// TwinCAT 3 PLC project ModBusPLC
// ProgramVersion: 3.1.4026.9
// libraries:
//   ModBus_For_FactoryIO, * (Kristian Zitny)
//   Tc2_ModbusSrv, * (Beckhoff Automation GmbH)
//   Tc2_Standard, * (Beckhoff Automation GmbH)
//   Tc2_System, * (Beckhoff Automation GmbH)
// project tree:
//   GVLs/ GVL_Factory_IO.TcGVL, GVL_IO.TcGVL
//   / PlcTask.TcTTO
//   POUs/Demonstration/ DemoProgram.TcPOU
//   POUs/Demonstration/DUTS/ E_FIO_PNP_State.TcDUT, ST_FIO_AxisConfig.TcDUT, ST_FIO_AxisIO.TcDUT
//   POUs/Demonstration/FunctionBlocks/ FB_Encoder.TcPOU, FB_FactoryIO_AxisAnalog.TcPOU, FB_FactoryIO_Conveyor.TcPOU, FB_FactoryIO_Lamp.TcPOU, FB_FactoryIO_PickPlace2Axis.TcPOU, FB_FactoryIO_Pusher.TcPOU, FB_Pick_Place.TcPOU, FB_PulseTrain.TcPOU
//   POUs/Factory_IO/ Connection.TcPOU, FB_IOMapper256.TcPOU
//   POUs/ MAIN.TcPOU
// real-time tasks:
//   TASK PlcTask: cycle T#10ms, priority 20, ADS port 350

CONFIGURATION ModBusPLC
    RESOURCE PLC ON TwinCAT3
        TASK PlcTask(INTERVAL := T#10ms, PRIORITY := 20);
        PROGRAM MAIN WITH PlcTask : MAIN;
    END_RESOURCE
END_CONFIGURATION

// ---- POUs/Demonstration/DUTS/E_FIO_PNP_State.TcDUT
TYPE E_FIO_PNP_State :
(
    Idle,
    MoveToPick,
    Grab,
    LiftAfterPick,
    MoveToPlace,
    Release,
    RetractAfterPlace,
    Error
);
END_TYPE

// ---- POUs/Demonstration/DUTS/ST_FIO_AxisConfig.TcDUT
TYPE ST_FIO_AxisConfig :
STRUCT
    MinPos     : LREAL;    // engineering units (e.g. mm)
    MaxPos     : LREAL;    // engineering units
    Tolerance  : LREAL;    // within tolerance -> in position
    Kp         : LREAL;    // proportional gain (engineering units per second)
    MaxVel     : LREAL;    // max velocity (engineering units per second)
END_STRUCT
END_TYPE

// ---- POUs/Demonstration/DUTS/ST_FIO_AxisIO.TcDUT
TYPE ST_FIO_AxisIO :
STRUCT
    SetPos : LREAL;   // output: position command to "analog output"
    ActPos : LREAL;   // input: feedback from "analog input"
END_STRUCT
END_TYPE

// ---- GVLs/GVL_Factory_IO.TcGVL
{attribute 'qualified_only'}
VAR_GLOBAL
	FIOinputs : ARRAY[0..31, 0..7] OF BOOL;
	FIOoutputs : ARRAY [0..255] OF BOOL;
END_VAR

// ---- GVLs/GVL_IO.TcGVL
{attribute 'qualified_only'}
VAR_GLOBAL
	Input : ARRAY [0..255] OF BOOL;
	Output : ARRAY [0..255] OF BOOL;
	AnalogInput : ARRAY [0..63] OF REAL;
	AnalogOutput : ARRAY [0..63] OF REAL;
END_VAR

// ---- POUs/MAIN.TcPOU
PROGRAM MAIN
VAR

END_VAR

// Call Connection Program for Connection with Factory IO Modbus Server //
Connection();
// Call Demo Program
DemoProgram();

END_PROGRAM

// ---- POUs/Factory_IO/Connection.TcPOU
PROGRAM Connection
VAR
	MB_Client: ModBus_For_Factory_IO;
	IO_Mapper: FB_IOMapper256;
END_VAR


	MB_Client(
	axInputs:= GVL_Factory_IO.FIOoutputs, 
	arInputs:= GVL_IO.AnalogOutput, 
	sIPaddr:= '127.0.0.1', 
	uiTCPPort:= 505, 
	iUnitID:= 1, 
	iNumberOfBoolInputs:= 256, 
	iNumberOfRegInputs:= 64, 
	iNumberOfBoolOutputs:= 256, 
	iNumberOfRegOutputs:= 64, 
	xStart:= TRUE, 
	axReaded=> GVL_Factory_IO.FIOinputs, 
	arReaded=> GVL_IO.AnalogInput, 
	xErrReadBoolFB=> , 
	udiErrNumberReadBoolFB=> , 
	sErrorDescriptionReadBoolFB=> , 
	xErrReadRegFB=> , 
	udiErrNumberReadRegFB=> , 
	sErrorDescriptionReadRegFB=> , 
	xErrWriteBoolFB=> , 
	udiErrNumberWriteBoolFB=> , 
	sErrorDescriptionWriteBoolFB=> , 
	xErrWriteRegFB=> , 
	udiErrNumberWriteRegFB=> , 
	sErrorDescriptionWriteRegFB=> );
	
	
	
	IO_Mapper(inputs:= GVL_Factory_IO.FIOinputs, outputs:= GVL_Factory_IO.FIOOutputs );

END_PROGRAM

// ---- POUs/Factory_IO/FB_IOMapper256.TcPOU
FUNCTION_BLOCK FB_IOMapper256
VAR_INPUT
    // Globale IO arrays
    inputs  : ARRAY [0..31, 0..7] OF BOOL;
END_VAR

VAR_IN_OUT
    outputs : ARRAY [0..255] OF BOOL;
END_VAR

VAR_OUTPUT
    
END_VAR

VAR
    i, j     : INT;
    flatIndex: INT;
END_VAR


// ===========================
// 1) Inputs 2D -> flat 0..255
// ===========================
FOR i := 0 TO 31 DO
    FOR j := 0 TO 7 DO
        flatIndex := i * 8 + j;
        GVL_IO.input[flatIndex] := inputs[i, j];
    END_FOR
END_FOR;


// ===========================
// 2) Outputs flat -> global
// ===========================
FOR flatIndex := 0 TO 255 DO
    outputs[flatIndex] := GVL_IO.Output[flatIndex];
END_FOR;

END_FUNCTION_BLOCK

// ---- POUs/Demonstration/DemoProgram.TcPOU
PROGRAM DemoProgram
VAR
	DemoEncoder_1: FB_Encoder;
	DemoEncoder_2: FB_Encoder;
	fEncoder1_Position: LREAL;
	fEncoder1_Velocity: LREAL;
	bEncoder1_Error: BOOL;
	nEncoder1_ErrorID: UINT;
	fEncoder2_Position: LREAL;
	fEncoder2_Velocity: LREAL;
	bEncoder2_Error: BOOL;
	nEncoder2_ErrorID: UINT;
	Start: BOOL;
	 
	ConvLeft: BOOL;
	ConvRight: BOOL;
	RotCW_1: BOOL;
	RotCCW_1: BOOL;
	Grab_1: BOOL;
	ProductSensorBlue: BOOL;
	ProductSensorGreen: BOOL;
	X_Cmd_1: REAL;
	Z_Cmd_1: REAL;
	X_Act_1: REAL;
	Z_Act_1: REAL;
	bXInPos_1: BOOL;
	bZInPos_1: BOOL;
	Sensor_ProductInFrontOfGripper: BOOL;
	LastKnownColour: STRING(INT#4);
	T_Grab_1: TON ;
	T_Rot_1: TON;
	T_Release_1: TON;
	T_EndTimer: TON;
	UseAdvancedMode: BOOL := TRUE;
	T_Rot_0: TON;
	ProductColour: REAL;
	T_Grab_2: TON;
	T_Rot_3: TON;
	T_Rot_4: TON;
	SafeX_1: REAL := 0;
END_VAR
VAR
    // -----------------------------
    // I/O mapping (adjust indices)
    // -----------------------------
    ProductSensor : BOOL;

    ConvAll : BOOL;

    RotCW  : BOOL;
    RotCCW : BOOL;
    Grab   : BOOL;

    // -----------------------------
    // "Analog" feedback/commands
    // -----------------------------
    X_Act : LREAL;
    Z_Act : LREAL;
    X_Cmd : LREAL;
    Z_Cmd : LREAL;

    // -----------------------------
    // Targets (demo values)
    // -----------------------------
    PickX  : LREAL := 6.0;
    PickZ  : LREAL := 10.0;

    PlaceX : LREAL := 7.0;
    PlaceZ : LREAL := 9.0;

    SafeZ  : LREAL := 0.0;
	
	PickX_1  : LREAL := 1.0;
    PickZ_1  : LREAL := 10.0;

    PlaceX_1 : LREAL := 10.0;
    PlaceZ_1 : LREAL := 10.0;

    SafeZ_1  : LREAL := 0.0;

    Tol    : LREAL := 1.0;

    // -----------------------------
    // State machine
    // -----------------------------
    State : INT := 0;
	StateAdvanced : INT := 0;

    // -----------------------------
    // Timers
    // -----------------------------
    T_Grab    : TON;
    T_Release : TON;
    T_Rot     : TON;

    // -----------------------------
    // Rotation pulse control
    // -----------------------------
    RotPulseActive : BOOL;

    // -----------------------------
    // Helpers
    // -----------------------------
    bXInPos : BOOL;
    bZInPos : BOOL;
END_VAR

VAR_INPUT
	
END_VAR

DemoEncoder_1(
	bEnable:= , 
	bA_Input:= GVL_IO.Input[8],
	bB_Input:= GVL_IO.Input[9], 
	bInvertDirection:= , 
	fUnitPerCount:= , 
	nVelSampleMs:= , 
	bRefSensor:= , 
	bRefCommand:= , 
	fRefPosition:= , 
	nCount=> , 
	fPosition=> fEncoder1_Position, 
	fVelocity=> fEncoder1_Velocity, 
	bReferenced=> , 
	bError=> bEncoder1_Error, 
	nErrorId=> nEncoder1_ErrorID);
	
	
	
										// =====================================================
										// Demo Program Simple Pick and Place
										// =====================================================	
		
	// =====================================================
	// Apply outputs (all 3 conveyors together)
	// =====================================================
	GVL_IO.Output[0] := ConvAll;
	GVL_IO.Output[1] := ConvAll;
	GVL_IO.Output[2] := ConvAll;
	GVL_IO.Output[4] := ConvAll;
	// Rotation interlock
	GVL_IO.Output[28] := RotCW ;
	GVL_IO.Output[29] := RotCCW ;
	
	// Grab
	GVL_IO.Output[3] := Grab;
	
	// Analog commands (map these to your Modbus registers / analog outputs)
	GVL_IO.AnalogOutput[0] := LREAL_TO_WORD(X_Cmd ); 
	GVL_IO.AnalogOutput[1] := LREAL_TO_WORD(Z_Cmd );
	

// =====================================================
// Read inputs (adjust mapping here)
// =====================================================
ProductSensor := GVL_IO.Input[7];
X_Act := GVL_IO.AnalogInput[0];
Z_Act := GVL_IO.AnalogInput[1];

// =====================================================
// Default outputs each scan
// =====================================================
//GVL_IO.Output[0] := FALSE; // conveyor 1
//GVL_IO.Output[1] := FALSE; // conveyor 2
//GVL_IO.Output[2] := FALSE; // conveyor 3

//RotCW := FALSE;
//RotCCW := FALSE;
Grab := FALSE;

// Rotation coils default off (interlock)



// Grab output default off
GVL_IO.Output[6] := FALSE; // grab

// Default hold current command
X_Cmd := X_Cmd;
Z_Cmd := Z_Cmd;

IF ConvAll THEN
	GVL_IO.Output[11] := TRUE; //Green Light
	GVL_IO.Output[10]:= FALSE;
	ELSE IF NOT ConvAll THEN
		GVL_IO.Output[10]:= TRUE; //Yellow Light
		GVL_IO.Output[11]:= FALSE;
	END_IF
END_IF

IF Connection.MB_Client.xErrReadBoolFB THEN 
	GVL_IO.Output[9] := TRUE; //Red Light
END_IF
// =====================================================
// Simple in-position checks (needs real feedback)
// =====================================================
bXInPos := (ABS(X_Cmd - X_Act) <= Tol);
bZInPos := (ABS(Z_Cmd - Z_Act) <= Tol);


// =====================================================
// State machine
// =====================================================
CASE State OF

// -----------------------------------------------------
// 0: conveyors on, wait product
// -----------------------------------------------------
0:
    ConvAll := TRUE;

	IF Sensor_ProductInFrontOfGripper THEN
        ConvAll := FALSE;
        State := 110;
    END_IF
	
    IF ProductSensor  THEN
        ConvAll := FALSE;
        State := 10;
    END_IF



// -----------------------------------------------------
// 10: move above pick (SafeZ + PickX)
// -----------------------------------------------------
10:
    ConvAll := FALSE;

    X_Cmd := PickX;
    Z_Cmd := SafeZ;

    IF (ABS(PickX - X_Act) <= Tol) AND (ABS(SafeZ - Z_Act) <= Tol) THEN
        State := 20;
    END_IF


// -----------------------------------------------------
// 20: go down to pick (PickZ)
// -----------------------------------------------------
20:
    ConvAll := FALSE;

    X_Cmd := PickX;
    Z_Cmd := PickZ;

    IF (ABS(PickZ - Z_Act) <= Tol) THEN
        State := 30;
    END_IF


// -----------------------------------------------------
// 30: grab for 0.5s
// -----------------------------------------------------
30:
    ConvAll := FALSE;

    X_Cmd := PickX;
    Z_Cmd := PickZ;

    Grab := TRUE;

    T_Grab(IN := TRUE, PT := T#250ms);
    IF T_Grab.Q THEN
        T_Grab(IN := FALSE);
        State := 40;
    END_IF


// -----------------------------------------------------
// 40: lift to SafeZ (keep grab)
// -----------------------------------------------------
40:
    ConvAll := FALSE;

    X_Cmd := PickX;
    Z_Cmd := SafeZ;

    Grab := TRUE;

    IF (ABS(SafeZ - Z_Act) <= Tol) THEN
        State := 50;
    END_IF


// -----------------------------------------------------
// 50: rotate CW pulse 0.5s (coil 4)
// -----------------------------------------------------
50:
    ConvAll := FALSE;

    X_Cmd := PickX;
    Z_Cmd := SafeZ;

    Grab := TRUE;

    GVL_IO.Output[50] := TRUE;

    T_Rot_0(IN := TRUE, PT := T#1500MS);
    IF T_Rot_0.Q THEN
        T_Rot_0(IN := FALSE);
        State := 60;
    END_IF


// -----------------------------------------------------
// 60: move above place (SafeZ + PlaceX)
// -----------------------------------------------------
60:
    ConvAll := FALSE;
	GVL_IO.Output[50] := FALSE;
    X_Cmd := PlaceX;
    Z_Cmd := SafeZ;

    Grab := TRUE;

    IF (ABS(PlaceX - X_Act) <= Tol) AND (ABS(SafeZ - Z_Act) <= Tol) THEN
        State := 70;
    END_IF


// -----------------------------------------------------
// 70: go down to place (PlaceZ)
// -----------------------------------------------------
70:
    ConvAll := FALSE;

    X_Cmd := PlaceX;
    Z_Cmd := PlaceZ;

    Grab := TRUE;

    IF (ABS(PlaceZ - Z_Act) <= Tol) THEN
        State := 80;
    END_IF


// -----------------------------------------------------
// 80: release and wait 1s
// -----------------------------------------------------
80:
    ConvAll := FALSE;

    X_Cmd := PlaceX;
    Z_Cmd := PlaceZ;

    Grab := FALSE;

    T_Release(IN := TRUE, PT := T#750MS);
    IF T_Release.Q THEN
        T_Release(IN := FALSE);
        State := 90;
    END_IF


// -----------------------------------------------------
// 90: lift again to SafeZ
// -----------------------------------------------------
90:
    ConvAll := FALSE;

    X_Cmd := PlaceX;
    Z_Cmd := SafeZ;

    Grab := FALSE;

    IF (ABS(SafeZ - Z_Act) <= Tol) THEN
        State := 100;
    END_IF


// -----------------------------------------------------
// 100: rotate CCW pulse 0.5s (coil 5)
// -----------------------------------------------------
100:
    ConvAll := FALSE;

    X_Cmd := PlaceX;
    Z_Cmd := SafeZ;

    Grab := FALSE;

    GVL_IO.Output[51] := TRUE;

    T_Rot(IN := TRUE, PT := T#400MS);
    IF T_Rot.Q THEN
        T_Rot(IN := FALSE);
        State := 110;
    END_IF


// -----------------------------------------------------
// 110: conveyors on again, wait sensor clear
// -----------------------------------------------------
110:
	GVL_IO.Output[51] := FALSE;
	IF NOT Sensor_ProductInFrontOfGripper THEN
		ConvAll := TRUE;
	END_IF
    

    IF NOT ProductSensor OR NOT Sensor_ProductInFrontOfGripper THEN
        State := 0;
    END_IF


ELSE
    State := 0;
END_CASE


											// =====================================================
											// Demo Program Advanced Pick and Place
											// =====================================================	
		
	// =====================================================
	// Apply outputs (all 3 conveyors together)
	// =====================================================
	GVL_IO.Output[14] := ConvLeft;
	GVL_IO.Output[15] := ConvLeft;
	GVL_IO.Output[16] := ConvLeft;
	GVL_IO.Output[17] := ConvLeft;
	GVL_IO.Output[18] := ConvLeft;
	GVL_IO.Output[19] := ConvLeft;
	GVL_IO.Output[20] := ConvLeft;
	GVL_IO.Output[21] := ConvRight;
	GVL_IO.Output[22] := ConvRight;
	GVL_IO.Output[23] := ConvRight;
	GVL_IO.Output[24] := ConvRight;
	GVL_IO.Output[25] := ConvRight;
	GVL_IO.Output[26] := ConvRight;
	GVL_IO.Output[27] := ConvRight;
	
	
	// Grab
	GVL_IO.Output[5] := Grab_1;
	
	// Analog commands (map these to your Modbus registers / analog outputs)
	GVL_IO.AnalogOutput[2] := LREAL_TO_WORD(X_Cmd_1 ); 
	GVL_IO.AnalogOutput[3] := LREAL_TO_WORD(Z_Cmd_1 );
	

// =====================================================
// Read inputs (adjust mapping here)
// =====================================================
ProductSensorBlue := GVL_IO.Input[12];
ProductSensorGreen := GVL_IO.Input[13];
Sensor_ProductInFrontOfGripper := GVL_IO.Input[6];
X_Act_1 := GVL_IO.AnalogInput[2];
Z_Act_1 := GVL_IO.AnalogInput[3];
ProductColour := GVL_IO.AnalogInput[4];


// =====================================================
// Default outputs each scan
// =====================================================
//GVL_IO.Output[0] := FALSE; // conveyor 1
//GVL_IO.Output[1] := FALSE; // conveyor 2
//GVL_IO.Output[2] := FALSE; // conveyor 3


Grab_1 := FALSE;
ConvLeft := FALSE;
ConvRight := FALSE;

// Default hold current command
X_Cmd_1 := X_Cmd_1;
Z_Cmd_1 := Z_Cmd_1;


// =====================================================
// Simple in-position checks (needs real feedback)
// =====================================================
bXInPos_1 := (ABS(X_Cmd_1 - X_Act_1) <= Tol);
bZInPos_1 := (ABS(Z_Cmd_1 - Z_Act_1) <= Tol);

// =====================================================
// Colour Helpers
// =====================================================

IF Connection.MB_Client.arReaded[4] = 0.1 THEN
    LastKnownColour := 'BLUE';
ELSIF Connection.MB_Client.arReaded[4] = 5 THEN
    LastKnownColour := 'GREEN';
END_IF

// =====================================================
// State machine
// =====================================================
IF UseAdvancedMode THEN
	
	CASE StateAdvanced OF
	
	// -----------------------------------------------------
	// 0: Start Cycle
	// -----------------------------------------------------
	0:
		IF Sensor_ProductInFrontOfGripper THEN
			StateAdvanced := 10;
		END_IF
		  
		
	
	// -----------------------------------------------------
	// 10: move above pick (SafeZ + PickX)
	// -----------------------------------------------------
	10:
		
	
		X_Cmd_1 := PickX_1;
		Z_Cmd_1 := SafeZ_1;
	
		IF (ABS(PickX_1 - X_Act_1) <= Tol) AND (ABS(SafeZ_1 - Z_Act_1) <= Tol) THEN
			StateAdvanced := 20;
		END_IF
	
	
	// -----------------------------------------------------
	// 20: go down to pick (PickZ)
	// -----------------------------------------------------
	20:
		
	
		X_Cmd_1 := PickX_1;
		Z_Cmd_1 := PickZ_1;
	
		IF (ABS(PickZ_1 - Z_Act_1) <= Tol) THEN
			StateAdvanced := 30;
		END_IF
	
	
	// -----------------------------------------------------
	// 30: grab for 0.5s
	// -----------------------------------------------------
	30:
		
	
		X_Cmd_1 := PickX_1;
		Z_Cmd_1 := PickZ_1;
	
		Grab_1 := TRUE;
	
		T_Grab_2(IN := TRUE, PT := T#250MS);
		IF T_Grab_2.Q THEN
			T_Grab_2(IN := FALSE);
			StateAdvanced := 40;
		END_IF
	
	
	// -----------------------------------------------------
	// 40: lift to SafeZ (keep grab)
	// -----------------------------------------------------
	40:
		
	
		X_Cmd_1 := PickX_1;
		Z_Cmd_1 := SafeZ_1;
	
		Grab_1 := TRUE;
		
		IF (ABS(SafeZ_1 - Z_Act_1) <= Tol) THEN
			StateAdvanced := 45;
		END_IF
	
	// -----------------------------------------------------
	// 45: Prepare move based on colour
	// -----------------------------------------------------
	45:
		
		IF LastKnownColour = 'BLUE' THEN
			StateAdvanced := 50;
		END_IF
		
		IF LastKnownColour = 'GREEN' THEN
			StateAdvanced := 55;
		END_IF
	
	// -----------------------------------------------------
	// 50: rotate CW pulse 0.5s (coil 4)
	// -----------------------------------------------------
	50:
		
	
		X_Cmd_1 := PickX_1;
		Z_Cmd_1 := SafeZ_1;
	
		Grab_1 := TRUE;
		ConvRight := FALSE;
		GVL_IO.Output[12] := TRUE;
	
		T_Rot_3(IN := TRUE, PT := T#1200MS);
		IF T_Rot_3.Q THEN
			T_Rot_3(IN := FALSE);
			StateAdvanced := 60;
		END_IF
	
	// -----------------------------------------------------
	// 55: rotate CCW pulse 0.5s (coil 4)
	// -----------------------------------------------------
	55:
		
		X_Cmd_1 := PickX_1;
		Z_Cmd_1 := SafeZ_1;
	
		Grab_1 := TRUE;
	
		GVL_IO.Output[13] := TRUE;
	
		T_Rot_4(IN := TRUE, PT := T#1200MS);
		IF T_Rot_4.Q THEN
			T_Rot_4(IN := FALSE);
			StateAdvanced := 60;
		END_IF
	
	
	// -----------------------------------------------------
	// 60: move above place (SafeZ + PlaceX)
	// -----------------------------------------------------
	60:
		GVL_IO.Output[12] := FALSE;
		GVL_IO.Output[13] := FALSE;
		X_Cmd_1 := PlaceX_1;
		Z_Cmd_1 := SafeZ_1;
	
		Grab_1 := TRUE;
	
		IF (ABS(PlaceX_1 - X_Act_1) <= Tol) AND (ABS(SafeZ_1 - Z_Act_1) <= Tol) THEN
			StateAdvanced := 70;
		END_IF
	
	
	// -----------------------------------------------------
	// 70: go down to place (PlaceZ)
	// -----------------------------------------------------
	70:
		
	
		X_Cmd_1 := PlaceX_1;
		Z_Cmd_1 := PlaceZ_1;
	
		Grab_1 := TRUE;
	
		IF (ABS(PlaceZ_1 - Z_Act_1) <= Tol) THEN
			StateAdvanced := 80;
		END_IF
	
	
	// -----------------------------------------------------
	// 80: release and wait 1s
	// -----------------------------------------------------
	80:
		
	
		X_Cmd_1 := PlaceX_1;
		Z_Cmd_1 := PlaceZ_1;
	
		Grab_1 := FALSE;
	
		T_Release_1(IN := TRUE, PT := T#750MS);
		IF T_Release_1.Q THEN
			T_Release_1(IN := FALSE);
			StateAdvanced := 90;
		END_IF
	
	
	// -----------------------------------------------------
	// 90: lift again to SafeZ
	// -----------------------------------------------------
	90:
		
	
		X_Cmd_1 := SafeX_1;
		Z_Cmd_1 := SafeZ_1;
	
		Grab_1 := FALSE;
	
		IF (ABS(SafeZ_1 - Z_Act_1) <= Tol) THEN
			StateAdvanced := 100;
		END_IF
	
	
	// -----------------------------------------------------
	// 100: SPARE Step
	// -----------------------------------------------------
	100:
		X_Cmd_1 := PickX_1;
		Z_Cmd_1 := SafeZ_1;
	
		Grab_1 := TRUE;
	
		GVL_IO.Output[13] := TRUE;
	
		T_Rot_4(IN := TRUE, PT := T#1200MS);
		IF T_Rot_4.Q THEN
			T_Rot_4(IN := FALSE);
			StateAdvanced := 110;
		END_IF
			
		
	
	
	// -----------------------------------------------------
	// 110: Start Conveyors
	// -----------------------------------------------------
	110:
		IF LastKnownColour = 'BLUE' THEN
			ConvRight := TRUE;
		END_IF
		
		IF LastKnownColour = 'GREEN' THEN
			ConvLeft := TRUE;
		END_IF
	
		T_EndTimer(IN := TRUE, PT := T#750MS);
		IF T_EndTimer.Q THEN
			T_EndTimer(IN := FALSE);
			StateAdvanced := 0;
		END_IF
			   
	
	
	ELSE
		StateAdvanced := 0;
	END_CASE
	
END_IF

END_PROGRAM

// ---- POUs/Demonstration/FunctionBlocks/FB_Encoder.TcPOU
FUNCTION_BLOCK FB_Encoder
VAR_INPUT
    bEnable         : BOOL := TRUE;

    bA_Input              : BOOL;
    bB_Input              : BOOL;

    bInvertDirection: BOOL := FALSE;

    fUnitPerCount   : LREAL := 1.0;     // engineering units per count (must be > 0)
    nVelSampleMs    : UINT  := 10;      // speed update interval in ms (e.g. 5..50)

    // Optional referencing
    bRefSensor      : BOOL := FALSE;    // e.g. IO_Control.DigitalInput[RefSensor_Index].bDesiredInput
    bRefCommand     : BOOL := FALSE;    // e.g. HMI button
    fRefPosition    : LREAL := 0.0;     // desired position when referencing happens
END_VAR

VAR_OUTPUT
    nCount      : DINT;     // raw counts
    fPosition   : LREAL;    // (nCount * fUnitPerCount) - fOffset
    fVelocity   : LREAL;    // units per second
    bReferenced : BOOL;

    bError      : BOOL;
    nErrorId    : UINT;
END_VAR

VAR
    // 1ms ticker / time base (no external libs)
    fbMsTicker      : TON;
    dwCurrentTimeMs : UDINT;
    dwPrevVelTimeMs : UDINT;

    // Quadrature decode
    byPrevAB : BYTE;
    byNowAB  : BYTE;

    // Velocity sampling
    nPrevVelCount : DINT;

    // Referencing
    rtRefSensor  : R_TRIG;
    rtRefCommand : R_TRIG;

    fOffset      : LREAL;

    // Internals
    nDelta       : DINT;
    fDirSign     : LREAL;
    dtMs         : UDINT;
END_VAR


// =====================================================
// Map your ref sensor like you requested (example line)
// =====================================================
// bRefSensor := IO_Control.DigitalInput[RefSensor_Index].bDesiredInput;


// =========================
// 0) Time base (1ms ticker)
// =========================
fbMsTicker(IN := TRUE, PT := T#1MS);

IF fbMsTicker.Q THEN
    fbMsTicker(IN := FALSE);
    fbMsTicker(IN := TRUE);

    IF dwCurrentTimeMs = 16#FFFFFFFF THEN
        dwCurrentTimeMs := 0;
    ELSE
        dwCurrentTimeMs := dwCurrentTimeMs + 1;
    END_IF
END_IF;


// ======================
// 1) Basic guards/default
// ======================
bError   := FALSE;
nErrorId := 0;

IF NOT bEnable THEN
    // No disable-state text/flags; just do nothing and keep last values
    RETURN;
END_IF;

IF fUnitPerCount <= 0.0 THEN
    bError   := TRUE;
    nErrorId := 1; // invalid scaling
    RETURN;
END_IF;

IF bInvertDirection THEN
    fDirSign := -1.0;
ELSE
    fDirSign := 1.0;
END_IF;


// ==================================
// 2) Quadrature A/B position counting
//    Valid sequence: 00 -> 01 -> 11 -> 10 -> 00 (and reverse)
// ==================================
byNowAB := 0;
IF bA_Input THEN byNowAB := byNowAB OR 1; END_IF;   // bit0 = A
IF bB_Input THEN byNowAB := byNowAB OR 2; END_IF;   // bit1 = B

IF byNowAB <> byPrevAB THEN
    // Transition table (prev -> now) gives delta in counts:
    // Forward: 00->01, 01->11, 11->10, 10->00  => +1
    // Reverse: 00->10, 10->11, 11->01, 01->00  => -1
    nDelta := 0;

    CASE byPrevAB OF
        0: // 00
            CASE byNowAB OF
                1: nDelta :=  1; // 00->01
                2: nDelta := -1; // 00->10
                ELSE nDelta := 0;
            END_CASE

        1: // 01
            CASE byNowAB OF
                3: nDelta :=  1; // 01->11
                0: nDelta := -1; // 01->00
                ELSE nDelta := 0;
            END_CASE

        3: // 11
            CASE byNowAB OF
                2: nDelta :=  1; // 11->10
                1: nDelta := -1; // 11->01
                ELSE nDelta := 0;
            END_CASE

        2: // 10
            CASE byNowAB OF
                0: nDelta :=  1; // 10->00
                3: nDelta := -1; // 10->11
                ELSE nDelta := 0;
            END_CASE
        ELSE
            nDelta := 0;
    END_CASE

    // If you want: flag invalid jumps (e.g. 00->11) as error
    IF nDelta = 0 THEN
        // invalid / bounce / skipped state
        bError   := TRUE;
        nErrorId := 2; // invalid AB transition
    ELSE
        // Apply direction sign
        IF fDirSign < 0.0 THEN
            nDelta := -nDelta;
        END_IF;

        nCount := nCount + nDelta;
    END_IF;

    byPrevAB := byNowAB;
END_IF;


// =============================
// 3) Position in engineering units
// =============================
fPosition := (DINT_TO_LREAL(nCount) * fUnitPerCount) - fOffset;


// =============================
// 4) Velocity (sampled every nVelSampleMs)
// =============================
IF dwPrevVelTimeMs = 0 THEN
    dwPrevVelTimeMs := dwCurrentTimeMs;
    nPrevVelCount   := nCount;
ELSE
    dtMs := dwCurrentTimeMs - dwPrevVelTimeMs;

    IF dtMs >= UINT_TO_UDINT(nVelSampleMs) THEN
        // units/s = (deltaCounts * unitPerCount) / (dtMs/1000)
        fVelocity := (DINT_TO_LREAL(nCount - nPrevVelCount) * fUnitPerCount) / (UDINT_TO_LREAL(dtMs) / 1000.0);

        dwPrevVelTimeMs := dwCurrentTimeMs;
        nPrevVelCount   := nCount;
    END_IF;
END_IF;


// =============================
// 5) Optional referencing (simple)
// =============================
rtRefSensor(CLK := bRefSensor);
rtRefCommand(CLK := bRefCommand);

// Reference on sensor rising edge
IF rtRefSensor.Q THEN
    fOffset     := (DINT_TO_LREAL(nCount) * fUnitPerCount) - fRefPosition;
    bReferenced := TRUE;
END_IF;

// Manual reference only allowed when sensor is active (optional rule)
IF rtRefCommand.Q THEN
    IF bRefSensor THEN
        fOffset     := (DINT_TO_LREAL(nCount) * fUnitPerCount) - fRefPosition;
        bReferenced := TRUE;
    ELSE
        bError   := TRUE;
        nErrorId := 3; // ref command without sensor
    END_IF;
END_IF;

END_FUNCTION_BLOCK

// ---- POUs/Demonstration/FunctionBlocks/FB_FactoryIO_AxisAnalog.TcPOU
FUNCTION_BLOCK FB_FactoryIO_AxisAnalog
VAR_INPUT
    Enable      : BOOL;
    TargetPos   : LREAL;
    ActualPos   : LREAL;

    MaxSpeed    : LREAL := 100;
    Tolerance   : LREAL := 1;

    CycleTime   : LREAL := 0.01;
	error : LREAL;
    step  : LREAL;
END_VAR

VAR_OUTPUT
    CmdPos      : LREAL;
    InPosition  : BOOL;
END_VAR


IF NOT Enable THEN
    CmdPos := ActualPos;
    InPosition := FALSE;
    RETURN;
END_IF

CmdPos := TargetPos;
InPosition := (ABS(TargetPos - ActualPos) <= Tolerance);

END_FUNCTION_BLOCK

// ---- POUs/Demonstration/FunctionBlocks/FB_FactoryIO_Conveyor.TcPOU
FUNCTION_BLOCK FB_FactoryIO_Conveyor
VAR_INPUT
    bStart      : BOOL;
    bStop       : BOOL;
    bSensor     : BOOL;
END_VAR

VAR_OUTPUT
    bMotor      : BOOL;
    bRunning    : BOOL;
    bProduct    : BOOL;
END_VAR

VAR
    bRun : BOOL;
END_VAR


// Run latch
IF bStart THEN
    bRun := TRUE;
END_IF

IF bStop THEN
    bRun := FALSE;
END_IF

bMotor := bRun;
bRunning := bRun;

// Product detect
bProduct := bSensor;

END_FUNCTION_BLOCK

// ---- POUs/Demonstration/FunctionBlocks/FB_FactoryIO_Lamp.TcPOU
FUNCTION_BLOCK FB_FactoryIO_Lamp
VAR_INPUT
    bOn : BOOL;
END_VAR

VAR_OUTPUT
    OutSignal : BOOL;
END_VAR

OutSignal := bOn;

END_FUNCTION_BLOCK

// ---- POUs/Demonstration/FunctionBlocks/FB_FactoryIO_PickPlace2Axis.TcPOU
FUNCTION_BLOCK FB_FactoryIO_PickPlace2Axis
VAR_INPUT

    Enable : BOOL;
    Start  : BOOL;

    PickX  : LREAL;
    PickZ  : LREAL;

    PlaceX : LREAL;
    PlaceZ : LREAL;

    SafeZ  : LREAL;

    ActX   : LREAL;
    ActZ   : LREAL;

    MaterialDetected : BOOL ;

	GrabTime : TIME := T#1500MS;   // time to "grab" at pick position
END_VAR


VAR_OUTPUT

    CmdX : LREAL;
    CmdZ : LREAL;

    Grab : BOOL;

    RotateCW : BOOL;

    Busy : BOOL;
    Done : BOOL;

    State : INT;
    Error : BOOL;
    ErrorText : STRING(80);
	
END_VAR


VAR
	TonGrab : TON;
    AxisX : FB_FactoryIO_AxisAnalog;
    AxisZ : FB_FactoryIO_AxisAnalog;

	TON_1: TON;
	ReleaseTimer : TON;
END_VAR

// Default outputs each cycle
Done := FALSE;
Error := FALSE;
ErrorText := '';


// Grab timer runs only in Grab state
TonGrab(IN := (State = 30), PT := GrabTime);


CASE State OF

// =================================================
0: // idle
// =================================================
    Busy := FALSE;
    Grab := FALSE;

    IF Enable AND Start THEN
        Busy := TRUE;
        State := 10;
    END_IF


// =================================================
10: // move above pick (SafeZ + PickX)
// =================================================
    Busy := TRUE;
    Grab := FALSE;

    AxisZ(
        Enable := TRUE,
        TargetPos := SafeZ,
        ActualPos := ActZ
    );

    AxisX(
        Enable := TRUE,
        TargetPos := PickX,
        ActualPos := ActX
    );

    CmdX := AxisX.CmdPos;
    CmdZ := AxisZ.CmdPos;

    IF AxisX.InPosition AND AxisZ.InPosition THEN
        State := 20;
    END_IF


// =================================================
20: // go down to pick (PickZ)
// =================================================
    Busy := TRUE;
    Grab := FALSE;

    AxisZ(
        Enable := TRUE,
        TargetPos := PickZ,
        ActualPos := ActZ
    );

    AxisX(
        Enable := TRUE,
        TargetPos := PickX,
        ActualPos := ActX
    );

    CmdX := AxisX.CmdPos;
    CmdZ := AxisZ.CmdPos;

    IF AxisZ.InPosition THEN
        State := 30;
    END_IF


// =================================================
30: // grab (wait GrabTime)
// =================================================
    Busy := TRUE;
    Grab := TRUE;

    // Hold position during grabbing
    AxisZ(
        Enable := TRUE,
        TargetPos := PickZ,
        ActualPos := ActZ
    );

    AxisX(
        Enable := TRUE,
        TargetPos := PickX,
        ActualPos := ActX
    );

    CmdX := AxisX.CmdPos;
    CmdZ := AxisZ.CmdPos;

    IF TonGrab.Q THEN
        State := 40;
    END_IF


// =================================================
40: // lift (SafeZ)
// =================================================
    Busy := TRUE;
    Grab := TRUE;

    AxisZ(
        Enable := TRUE,
        TargetPos := SafeZ,
        ActualPos := ActZ
    );

    AxisX(
        Enable := TRUE,
        TargetPos := PickX,
        ActualPos := ActX
    );

    CmdX := AxisX.CmdPos;
    CmdZ := AxisZ.CmdPos;

    IF AxisZ.InPosition THEN
        State := 50;
    END_IF


// =================================================
50: // move to place X (PlaceX) at SafeZ
// =================================================
    Busy := TRUE;
    Grab := TRUE;

    AxisZ(
        Enable := TRUE,
        TargetPos := SafeZ,
        ActualPos := ActZ
    );

    AxisX(
        Enable := TRUE,
        TargetPos := PlaceX,
        ActualPos := ActX
    );

    CmdX := AxisX.CmdPos;
    CmdZ := AxisZ.CmdPos;

    IF AxisX.InPosition AND AxisZ.InPosition THEN
        State := 60;
    END_IF


// =================================================
60: // go down to place (PlaceZ)
// =================================================
    Busy := TRUE;
    Grab := TRUE;

    AxisZ(
        Enable := TRUE,
        TargetPos := PlaceZ,
        ActualPos := ActZ
    );

    AxisX(
        Enable := TRUE,
        TargetPos := PlaceX,
        ActualPos := ActX
    );

    CmdX := AxisX.CmdPos;
    CmdZ := AxisZ.CmdPos;

    IF AxisZ.InPosition THEN
        State := 70;
    END_IF


// =================================================
70: // release
// =================================================

Busy := TRUE;
Grab := FALSE;

// start timer
ReleaseTimer(IN := TRUE, PT := T#1S);

IF ReleaseTimer.Q THEN

    ReleaseTimer(IN := FALSE);

    State := 80;

END_IF

// =================================================
80: // lift again (SafeZ) and finish
// =================================================
    Busy := TRUE;
    Grab := FALSE;

    AxisZ(
        Enable := TRUE,
        TargetPos := SafeZ,
        ActualPos := ActZ
    );

    AxisX(
        Enable := TRUE,
        TargetPos := PlaceX,
        ActualPos := ActX
    );

    CmdX := AxisX.CmdPos;
    CmdZ := AxisZ.CmdPos;

    IF AxisZ.InPosition THEN
        Done := TRUE;
        Busy := FALSE;
        State := 0;
    END_IF


ELSE
    // Fallback
    Error := TRUE;
    ErrorText := 'Invalid state';
    State := 0;
END_CASE

END_FUNCTION_BLOCK

// ---- POUs/Demonstration/FunctionBlocks/FB_FactoryIO_Pusher.TcPOU
FUNCTION_BLOCK FB_FactoryIO_Pusher
VAR_INPUT
    bPushCmd      : BOOL;
    bRetractCmd   : BOOL;
    bExtendedSens : BOOL;
    bRetractedSens: BOOL;
END_VAR

VAR_OUTPUT
    bExtend       : BOOL;
    bRetract      : BOOL;
    bBusy         : BOOL;
END_VAR

VAR
    state : INT;
END_VAR

CASE state OF

0: // idle
    bBusy := FALSE;

    IF bPushCmd THEN
        state := 10;
    END_IF

10: // extend
    bExtend := TRUE;
    bRetract := FALSE;
    bBusy := TRUE;

    IF bExtendedSens THEN
        state := 20;
    END_IF

20: // retract
    bExtend := FALSE;
    bRetract := TRUE;

    IF bRetractedSens THEN
        state := 0;
    END_IF

END_CASE

END_FUNCTION_BLOCK

// ---- POUs/Demonstration/FunctionBlocks/FB_Pick_Place.TcPOU
FUNCTION_BLOCK FB_Pick_Place
VAR_INPUT
    Enable   : BOOL;
    Start    : BOOL; // pulse (1 cycle)
    Reset    : BOOL;

    PickX  : LREAL;
    PickZ  : LREAL;
    PlaceX : LREAL;
    PlaceZ : LREAL;
    SafeZ  : LREAL;

    ActX   : LREAL;
    ActZ   : LREAL;

    GrabTime : TIME := T#500ms;
END_VAR

VAR_OUTPUT
    CmdX : LREAL;
    CmdZ : LREAL;

    Grab : BOOL;

    Busy : BOOL;
    Done : BOOL;
    Error : BOOL;
    ErrorText : STRING(80);

    State : INT;
	bRotateCmd : BOOL;
	bRotateCmdCCW : BOOL;
END_VAR

VAR
    AxisX : FB_FactoryIO_AxisAnalog;
    AxisZ : FB_FactoryIO_AxisAnalog;

    StartTrig : R_TRIG;
    TonGrab : TON;
    TonRelease : TON;
	 Rot1 : FB_PulseTrain;
    Rot3 : FB_PulseTrain;
END_VAR

// Reset
IF Reset THEN
    State := 0;
    Busy := FALSE;
    Done := FALSE;
    Error := FALSE;
    ErrorText := '';
END_IF

Done := FALSE;
Error := FALSE;
ErrorText := '';

StartTrig(CLK := Start);

// Grab timer only in grab state
TonGrab(IN := (State = 30), PT := GrabTime);

// Release delay 1s in release state (optional, you wanted this)
TonRelease(IN := (State = 70), PT := T#1S);

CASE State OF

0: // idle
    Busy := FALSE;
    Grab := FALSE;

    // Hold current position
    AxisX(Enable := FALSE, TargetPos := ActX, ActualPos := ActX);
    AxisZ(Enable := FALSE, TargetPos := ActZ, ActualPos := ActZ);
    CmdX := ActX;
    CmdZ := ActZ;

    IF Enable AND StartTrig.Q THEN
        Busy := TRUE;
        State := 10;
    END_IF

10: // move above pick (SafeZ + PickX)
    Busy := TRUE;
    Grab := FALSE;

    AxisZ(Enable := TRUE, TargetPos := SafeZ, ActualPos := ActZ);
    AxisX(Enable := TRUE, TargetPos := PickX, ActualPos := ActX);

    CmdX := AxisX.CmdPos;
    CmdZ := AxisZ.CmdPos;

    IF AxisX.InPosition AND AxisZ.InPosition THEN
        State := 20;
    END_IF

20: // go down to pick (PickZ)
    Busy := TRUE;
    Grab := FALSE;

    AxisZ(Enable := TRUE, TargetPos := PickZ, ActualPos := ActZ);
    AxisX(Enable := TRUE, TargetPos := PickX, ActualPos := ActX);

    CmdX := AxisX.CmdPos;
    CmdZ := AxisZ.CmdPos;

    IF AxisZ.InPosition THEN
        State := 30;
    END_IF

30: // grab (wait GrabTime)
    Busy := TRUE;
    Grab := TRUE;

    AxisZ(Enable := TRUE, TargetPos := PickZ, ActualPos := ActZ);
    AxisX(Enable := TRUE, TargetPos := PickX, ActualPos := ActX);

    CmdX := AxisX.CmdPos;
    CmdZ := AxisZ.CmdPos;

    IF TonGrab.Q THEN
        State := 40;
    END_IF

40: // lift (SafeZ)
    Busy := TRUE;
    Grab := TRUE;

    AxisZ(Enable := TRUE, TargetPos := SafeZ, ActualPos := ActZ);
    AxisX(Enable := TRUE, TargetPos := PickX, ActualPos := ActX);

    CmdX := AxisX.CmdPos;
    CmdZ := AxisZ.CmdPos;

    IF AxisZ.InPosition THEN
        State := 41;
    END_IF
	
41: // ROTATE 1x 90° (only when robot done)
    Rot1(
        Enable := TRUE,
        PulseTime := T#500ms,
        PauseTime := T#500ms,
        Count := 1
    );

    bRotateCmd := Rot1.Q;

    IF Rot1.Done THEN
        State := 50;
    END_IF

50: // move to place X at SafeZ
    Busy := TRUE;
    Grab := TRUE;

    AxisZ(Enable := TRUE, TargetPos := SafeZ, ActualPos := ActZ);
    AxisX(Enable := TRUE, TargetPos := PlaceX, ActualPos := ActX);

    CmdX := AxisX.CmdPos;
    CmdZ := AxisZ.CmdPos;

    IF AxisX.InPosition AND AxisZ.InPosition THEN
        State := 60;
    END_IF

60: // go down to place (PlaceZ)
    Busy := TRUE;
    Grab := TRUE;

    AxisZ(Enable := TRUE, TargetPos := PlaceZ, ActualPos := ActZ);
    AxisX(Enable := TRUE, TargetPos := PlaceX, ActualPos := ActX);

    CmdX := AxisX.CmdPos;
    CmdZ := AxisZ.CmdPos;

    IF AxisZ.InPosition THEN
        State := 70;
    END_IF

70: // release + wait 1s
    Busy := TRUE;
    Grab := FALSE;

    // Hold position during release delay
    AxisZ(Enable := TRUE, TargetPos := PlaceZ, ActualPos := ActZ);
    AxisX(Enable := TRUE, TargetPos := PlaceX, ActualPos := ActX);

    CmdX := AxisX.CmdPos;
    CmdZ := AxisZ.CmdPos;

    IF TonRelease.Q THEN
        State := 80;
    END_IF

80: // lift again (SafeZ) and finish
    Busy := TRUE;
    Grab := FALSE;

    AxisZ(Enable := TRUE, TargetPos := SafeZ, ActualPos := ActZ);
    AxisX(Enable := TRUE, TargetPos := PlaceX, ActualPos := ActX);

    CmdX := AxisX.CmdPos;
    CmdZ := AxisZ.CmdPos;

    IF AxisZ.InPosition THEN
        Done := TRUE;
        Busy := FALSE;
        State := 90;
    END_IF
90: // Move CCW Back
    Rot3(
        Enable := TRUE,
        PulseTime := T#500ms,
        PauseTime := T#500ms,
        Count := 1
    );

    bRotateCmdCCW := Rot3.Q;

    IF Rot3.Done THEN
        State := 0;
    END_IF

ELSE
    Error := TRUE;
    ErrorText := 'Invalid state';
    Busy := FALSE;
    State := 0;
END_CASE

END_FUNCTION_BLOCK

// ---- POUs/Demonstration/FunctionBlocks/FB_PulseTrain.TcPOU
FUNCTION_BLOCK FB_PulseTrain
VAR_INPUT
    Enable     : BOOL;
    PulseTime  : TIME := T#500ms;
    PauseTime  : TIME := T#500ms;
    Count      : INT := 1;      // number of pulses
END_VAR

VAR_OUTPUT
    Q       : BOOL;  // output pulse signal
    Busy    : BOOL;
    Done    : BOOL;
END_VAR

VAR
    t : TON;
    phasePulse : BOOL;
    counter : INT;
END_VAR

IF NOT Enable THEN
    Q := FALSE;
    Busy := FALSE;
    Done := FALSE;
    t(IN := FALSE);
    phasePulse := TRUE;
    counter := 0;
    RETURN;
END_IF

Busy := TRUE;
Done := FALSE;

IF phasePulse THEN
    Q := TRUE;
    t(IN := TRUE, PT := PulseTime);
ELSE
    Q := FALSE;
    t(IN := TRUE, PT := PauseTime);
END_IF

IF t.Q THEN
    t(IN := FALSE);

    IF phasePulse THEN
        // pulse finished
        counter := counter + 1;
        phasePulse := FALSE;
    ELSE
        // pause finished
        phasePulse := TRUE;
    END_IF
END_IF

IF counter >= Count THEN
    Q := FALSE;
    Busy := FALSE;
    Done := TRUE;
END_IF

END_FUNCTION_BLOCK
